PROGRAM MAIN
VAR
	
END_VAR

END_PROGRAM

(* stored: Version 1.1.0.1, ProductVersion 3.1.4024.12
   POU MAIN: Id {f24a42c3-b030-4992-be5e-c24c89fa021d}, SpecialFunc None *)
